(* Logix 5000 project; controller SS1 Emulate 5570 rev 36.11; software revision 36.00 *)

TASK MainTask (continuous, watchdog 500 ms) : MainProgram

MODULES
   Local : Emulate 5570 (ICP 2, rev 36.11)
       : 1756-IB16 (ICP 3, rev 3.1, Input RPI 20 ms)
       : vendor 1 type 7 code 16 (ICP 4, rev 3.1, Output RPI 20 ms)
END_MODULES

VAR_GLOBAL   (* controller tags *)
   MOTOR : ALIAS FOR Local:4:O.Data.2;   // Motor Control
   PL1_OFF : ALIAS FOR Local:4:O.Data.0;   // Pilot Light 1 OFF (RED)
   PL2_ON : ALIAS FOR Local:4:O.Data.1;   // Pilot Light 1 ON (GREEN)
   START : ALIAS FOR Local:3:I.Data.1;   // Pushbutton Momentary N.O.
   STOP : ALIAS FOR Local:3:I.Data.0;   // Pushbutton Momentary N.C.
END_VAR

PROGRAM MainProgram   (* main routine MainFunction *)
VAR
   BAND_01 : FBD_BOOLEAN_AND := (In1 := 1, In2 := 1, In3 := 1, In4 := 1, In5 := 1, In6 := 1, In7 := 1, In8 := 1);   // AND For STOP PUSHBUTTON Holding Circuit
   BNOT_01 : FBD_BOOLEAN_NOT := (In := 1);   // OR for START Pushbutton Holding Circuit
   BOR_01 : FBD_BOOLEAN_OR;   // Invert for PL1_OFF Pilot Light
END_VAR

ROUTINE MainFunction   (* function block diagram *)
   SHEET 1
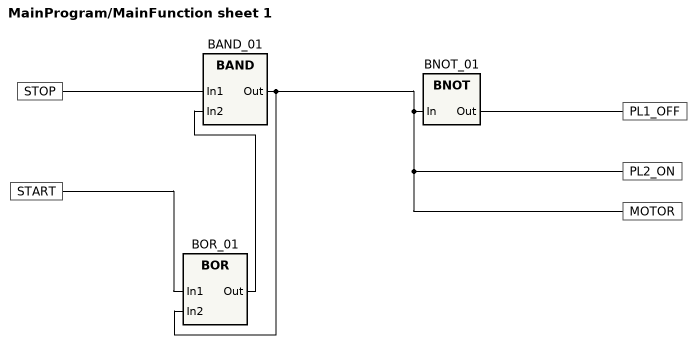
   BOR_01 : BOR(In1 := START, In2 := BAND_01.Out {feedback});
   BAND_01 : BAND(In1 := STOP, In2 := BOR_01.Out);
   BNOT_01 : BNOT(In := BAND_01.Out);
   PL1_OFF := BNOT_01.Out;
   PL2_ON := BAND_01.Out;
   MOTOR := BAND_01.Out;
END_ROUTINE
END_PROGRAM
